INTERFACE I_StationBehaviour

PROPERTY MoverVelocity : mc_lreal
GET
END_GET
SET
END_SET
END_PROPERTY

METHOD Reset : HRESULT
VAR_INPUT
END_VAR
END_METHOD

METHOD StartIndexing : BOOL
VAR_INPUT
END_VAR
END_METHOD

METHOD StopIndexing : BOOL
VAR_INPUT
END_VAR
END_METHOD

END_INTERFACE

(* stored: Version 1.1.0.1
   Itf I_StationBehaviour: Id {c83df270-a09e-429e-ad85-91c05aa15849}
   Property MoverVelocity: Id {5317f276-6413-492d-9d21-d374946fdc4f}
   Get Get: Id {21401961-8bae-4b54-8143-993acfe2699e}
   Set Set: Id {d4e38f48-028a-4774-a1cb-ef0b28a48b61}
   Method Reset: Id {ed2e6068-85fb-4db3-9ead-09d65d3faecc}
   Method StartIndexing: Id {9d162004-44cf-4117-bb96-7d190fd73fab}
   Method StopIndexing: Id {9953e0e8-7677-458f-a571-6742b50d758e} *)
